{attribute addProperty ShortName ""}
FUNCTION_BLOCK ABSTRACT CUBase EXTENDS TcoCore.TcoObject IMPLEMENTS ICuBase
VAR
    _statusInfo : CUBaseStatusInfo := (Parent := THIS^);
END_VAR

PROPERTY ABSTRACT Automat : REFERENCE TO TcoTaskedSequencer
GET
END_GET
END_PROPERTY

PROPERTY ABSTRACT Ground : REFERENCE TO TcoTaskedSequencer
GET
END_GET
END_PROPERTY

PROPERTY ABSTRACT Manual : REFERENCE TO TcoTaskedService
GET
END_GET
END_PROPERTY

PROPERTY ABSTRACT ProcessDataManager : REFERENCE TO ProcessDataManager
GET
END_GET
END_PROPERTY

METHOD UpdateInfo : BOOL
VAR_INPUT
END_VAR
IF Automat.Task.Busy THEN
    _statusInfo.Mode                   := eCUMode.AutomatMode;
    _statusInfo.CurrentTaskDescription := '<#AUTOMAT#>';
    _statusInfo.CurrentCycleTime       := Automat._SequenceElapsedTime;
    _statusInfo.CurrentUid             := Automat.CurrentStep.ID;
    _statusInfo.CurrentOperation       := Automat.CurrentStep.Description;
    _statusInfo.CurrentIsInStepMode    := Automat._modeController._mode = eSequencerMode.StepMode;
ELSIF Ground.Task.Busy THEN
    _statusInfo.Mode := eCUMode.GroundMode;
	_statusInfo.CurrentTaskDescription := '<#GROUND#>';
    _statusInfo.CurrentCycleTime       := Ground._SequenceElapsedTime;
    _statusInfo.CurrentUid             := Ground.CurrentStep.ID;
    _statusInfo.CurrentOperation       := Ground.CurrentStep.Description;
    _statusInfo.CurrentIsInStepMode    := Ground._modeController._mode = eSequencerMode.StepMode;
ELSIF THIS^.Manual.Busy THEN
    _statusInfo.Mode := eCUMode.ManualMode;
	_statusInfo.CurrentTaskDescription := '<#MANUAL#>';
ELSIF THIS^.Ground.Task.Done THEN
	_statusInfo.CurrentTaskDescription := '<#READY TO START#>';
	_statusInfo.Mode := eCUMode.GroundModeDone;
	_statusInfo.CurrentCycleTime       := Ground._SequenceElapsedTime;
    _statusInfo.CurrentUid             := Ground.CurrentStep.ID;
    _statusInfo.CurrentOperation       := Ground.CurrentStep.Description;
    _statusInfo.CurrentIsInStepMode    := Ground._modeController._mode = eSequencerMode.StepMode;
ELSE
    _statusInfo.Mode := eCUMode.NoMode;	
	_statusInfo.CurrentTaskDescription := '<#IDLE#>';
	_statusInfo.CurrentCycleTime       := T#0S;
    _statusInfo.CurrentUid             := 0;
    _statusInfo.CurrentOperation       := '';
    _statusInfo.CurrentIsInStepMode    := FALSE;
END_IF
END_METHOD

END_FUNCTION_BLOCK

(* stored: Version 1.1.0.1, ProductVersion 3.1.4024.9
   POU CUBase: Id {7de2193c-318e-4c64-a9a6-ba23fb2e4da1}, SpecialFunc None
   Property Automat: Id {9a1989f3-7511-4b12-80ce-78bb1add06c6}
   Get Get: Id {86426d31-47b7-4512-bf28-f740d21d447d}
   Property Ground: Id {6cf29f50-dec8-49c6-a97a-8a93927ca757}
   Get Get: Id {41f5a2de-fade-47b5-8a6c-d888d0eac9c5}
   Property Manual: Id {a2025997-47b5-45e1-80f0-0c1e8cce860d}
   Get Get: Id {c93ae827-0df1-40b0-b0fa-7bfc00959641}
   Property ProcessDataManager: Id {95e82431-3124-4f70-be63-551f0ca81c55}
   Get Get: Id {75873f97-0e26-4094-bf28-402fb0488241}
   Method UpdateInfo: Id {d2563fa9-29cd-48cb-9533-a53a49a45068} *)
